// TwinCAT 3 PLC project main
// ProgramVersion: 3.1.4024.0
// libraries:
//   Tc2_Math, * (Beckhoff Automation GmbH)
//   Tc2_Standard, * (Beckhoff Automation GmbH)
//   Tc2_System, * (Beckhoff Automation GmbH)
//   Tc3_Module, * (Beckhoff Automation GmbH)
//   Title, * (HSLU)
// project tree:
//   / PlcTask.TcTTO
//   POUs/ MAIN.TcPOU
// real-time tasks:
//   TASK PlcTask: cycle T#1ms, priority 20, ADS port 350

CONFIGURATION main
    RESOURCE PLC ON TwinCAT3
        TASK PlcTask(INTERVAL := T#1ms, PRIORITY := 20);
        PROGRAM MAIN WITH PlcTask : MAIN;
    END_RESOURCE
END_CONFIGURATION

// ---- POUs/MAIN.TcPOU
PROGRAM MAIN
VAR
	t :					REAL := 0;
	PWMValue025 :		REAL := 0;
	PWMValue05 :		REAL := 0;
	PWMValue075 :		REAL := 0;
	Integrator025 :		Integrator;
	Integrator05 : 		Integrator;
	Integrator075 :		Integrator;
	
	SinusValue10 :		REAL := 0;
	SinusValue1 :		REAL := 0;
	SinusValue100 :		REAL := 0;
	
	SquareValue :		REAL := 0;
	PT1 :				Tiefpassfilter;
	PT2 :				SecondOrderLag;
END_VAR

PWMValue025 := PwmSignal(ymin:= 0, ymax := 1, w:= 1, yoff:= 0, t:=t, PWM:= 0.25);
PWMValue05 := PwmSignal(ymin:= 0, ymax := 1, w:= 1, yoff:= 0, t:=t, PWM:= 0.5);
PWMValue075 := PwmSignal(ymin:= 0, ymax := 1, w:= 1, yoff:= 0, t:=t, PWM:= 0.75);
Integrator025(x:= PWMValue025, h:=0.001);
Integrator05(x:= PWMValue05, h:=0.001);
Integrator075(x:= PWMValue075, h:=0.001);

SinusValue10 := SinusFunction(A:=1,yoff:=0,w:=10,t:=t);
SinusValue1 := SinusFunction(A:=1,yoff:=0,w:=1,t:=t);
SinusValue100 := SinusFunction(A:=1,yoff:=0,w:=100,t:=t);

SquareValue := SquareSignal(ymin:= -1, ymax:= 1, w:= 10, yoff:= 0, t:=t);
PT1(x:=SquareValue,h:= 0.001,tau:= 0.1);
PT2(d:=0.2,w:=10,h:=0.001,x:=SquareValue);

t := t + 0.001;

END_PROGRAM
